TYPE ST_AxisStatus :
STRUCT
    fActualPosition : LREAL;
    fActualVelocity : LREAL;
    fActualTorque : LREAL;
    eAxisState : E_AxisState;
    bEnabled : BOOL;
    bHomed : BOOL;
    bInMotion : BOOL;
    bError : BOOL;
    nErrorCode : UDINT;
    bPositiveLimitActive : BOOL;
    bNegativeLimitActive : BOOL;
END_STRUCT
END_TYPE

(* stored: Version 1.1.0.1
   DUT ST_AxisStatus: Id {111F46E5-27DE-BDCB-3A42-332BA8E5DF5F} *)
